(* IEC 61131-3 sources: Fosela-House-/control/lib, 8 files *)

(* ---- Types_Common.st ---- *)
(* ============================================================
   Types_Common.st
   Tipos, enumeraciones y constantes compartidos entre
   FREE Smart (solar) y FREE Evolution (sistema principal).
   Proyecto: Fusela House — Jerez de la Frontera
   ============================================================ *)

(* ------------------------------------------------------------
   ENUMERACIONES
   ------------------------------------------------------------ *)

(* Modos del subsistema solar *)
TYPE E_Solar_Mode :
(
    SOLAR_AUTO      := 0,   (* Lógica automática según temperaturas *)
    SOLAR_FORCE_ACS := 1,   (* Forzar desvío a ACS *)
    SOLAR_FORCE_POOL:= 2,   (* Forzar desvío a piscina *)
    SOLAR_OFF       := 3    (* Solar desactivado *)
);
END_TYPE

(* Destino del primario de la BDC *)
TYPE E_BDC_Mode :
(
    BDC_OFF         := 0,
    BDC_ACS         := 1,   (* V3V1→D2 *)
    BDC_CLIMATE     := 2,   (* V3V1→V3V2→D3 *)
    BDC_POOL        := 3    (* V3V1→V3V2→HX_BDC *)
);
END_TYPE

(* Destino del HTR *)
TYPE E_HTR_Mode :
(
    HTR_ACS         := 0,   (* V3V3→serp.sup D2 (por defecto) *)
    HTR_POOL        := 1    (* V3V3→HX_HTR *)
);
END_TYPE

(* Estado de válvula de 3 vías *)
TYPE E_Valve3Way_Pos :
(
    V3W_POS_A       := 0,   (* Posición A (desenergizada / muelle) *)
    V3W_POS_B       := 1    (* Posición B (energizada) *)
);
END_TYPE

(* Modo de apartamento *)
TYPE E_Apartment_Mode :
(
    APT_PRECALENTADA := 0,  (* Alimenta CE desde agua precalentada (por defecto) *)
    APT_AFS          := 1   (* Alimenta CE desde AFS directa *)
);
END_TYPE

(* Fases del ciclo de pasteurización *)
TYPE E_Pasteurization_Phase :
(
    PAST_IDLE        := 0,  (* Sin ciclo activo *)
    PAST_HEAT_D2     := 1,  (* Calentando D2 a 70 °C *)
    PAST_HOLD_D2     := 2,  (* Manteniendo D2 ≥ 70 °C durante t_hold *)
    PAST_FLUSH_APT   := 3,  (* Purgado secuencial de apartamentos *)
    PAST_DONE        := 4   (* Ciclo completado *)
);
END_TYPE

(* Prioridad de la BDC *)
TYPE E_BDC_Priority :
(
    PRIO_ACS_CLIMATE_POOL := 0,  (* ACS > Climatización > Piscina *)
    PRIO_ACS_POOL_CLIMATE := 1   (* ACS > Piscina > Climatización *)
);
END_TYPE

(* ------------------------------------------------------------
   ESTRUCTURAS
   ------------------------------------------------------------ *)

(* Datos del subsistema solar publicados por FREE Smart *)
TYPE ST_SolarData :
STRUCT
    TT1             : REAL;     (* Temperatura colector [°C] *)
    TT2             : REAL;     (* D1 fondo [°C] *)
    TT3             : REAL;     (* D1 cabeza [°C] *)
    DT_solar        : REAL;     (* ΔT medido TT1-TT2 [K] *)
    vel_P1          : UINT;     (* Velocidad P1 [0-1000 ‰] *)
    pos_V3V_SOL     : BOOL;     (* FALSE=ACS, TRUE=piscina *)
    persianas_cerradas : BOOL;
    P2_activo       : BOOL;
    alarma_solar    : UINT;     (* 0=OK, ver códigos *)
    comm_ok         : BOOL;     (* Comunicación Modbus activa *)
END_STRUCT
END_TYPE

(* Alarmas del sistema *)
TYPE ST_SystemAlarms :
STRUCT
    (* Solar *)
    ALM_TT1_HIGH        : BOOL;  (* TT1 > ALM_TT1_MAX *)
    ALM_TT2_HIGH        : BOOL;  (* TT2 > ALM_TT2_MAX *)
    ALM_COMM_SMART      : BOOL;  (* Pérdida comunicación FREE Smart *)
    (* ACS *)
    ALM_TT5_LOW         : BOOL;  (* D2 cabeza por debajo de mínimo *)
    ALM_TT5_HIGH        : BOOL;  (* D2 sobretemperatura *)
    (* Piscina *)
    ALM_PISC_FLUJO      : BOOL;  (* IF_PISC sin flujo durante calentamiento *)
    ALM_PISC_T_HIGH     : BOOL;  (* TT11 > máximo piscina *)
    (* Climatización *)
    ALM_INUNDACION      : BOOL;  (* Sensor inundación bandeja fancoil *)
    ALM_D3_HIGH         : BOOL;  (* D3 sobretemperatura *)
    (* General *)
    ALM_BDC_FAULT       : BOOL;  (* Fallo BDC (entrada digital) *)
    CUALQUIER_ALARMA    : BOOL;  (* OR de todas *)
END_STRUCT
END_TYPE

(* ------------------------------------------------------------
   CONSTANTES — TEMPERATURAS (°C)
   ------------------------------------------------------------ *)
VAR_GLOBAL CONSTANT

    (* Solar *)
    C_SOLAR_DT_START    : REAL := 6.0;   (* ΔT arranque P1 *)
    C_SOLAR_DT_STOP     : REAL := 3.0;   (* ΔT parada P1 *)
    C_SOLAR_DT_TARGET   : REAL := 8.0;   (* ΔT objetivo lazo PI *)
    C_SOLAR_TT3_POOL    : REAL := 75.0;  (* TT3 mínimo para desvío a piscina *)
    C_SOLAR_TT1_MAX     : REAL := 95.0;  (* Alarma sobretemperatura colector *)
    C_SOLAR_TT2_DISS    : REAL := 85.0;  (* TT2 máximo antes de disipación *)
    C_SOLAR_TT2_LEGIONELLA : REAL := 45.0; (* Si TT2 lleva días por debajo → arranque forzado *)

    (* ACS *)
    C_ACS_TT4_START     : REAL := 50.0;  (* TT4 D2 fondo — arranque carga BDC *)
    C_ACS_TT4_STOP      : REAL := 55.0;  (* TT4 D2 fondo — parada carga BDC *)
    C_ACS_TT5_TARGET    : REAL := 65.0;  (* TT5 D2 cabeza — setpoint ACS *)
    C_ACS_TT5_HYST      : REAL := 3.0;   (* Histéresis TT5 *)
    C_ACS_VMT1          : REAL := 55.0;  (* Temperatura VMT1 [°C] — ajuste físico *)
    C_ACS_PAST_TARGET   : REAL := 70.0;  (* Temperatura pasteurización D2 *)
    C_ACS_PAST_HYST     : REAL := 2.0;   (* Histéresis pasteurización *)
    C_ACS_HTR_TT5_STOP  : REAL := 68.0;  (* TT5 que inhibe HTR hacia D2 *)

    (* Climatización *)
    C_CLIM_HEAT_START   : REAL := 45.0;  (* TT6 D3 arranque calefacción BDC *)
    C_CLIM_HEAT_STOP    : REAL := 50.0;  (* TT6 D3 parada calefacción *)
    C_CLIM_COOL_START   : REAL := 9.0;   (* TT7 D3 arranque refrigeración *)
    C_CLIM_COOL_STOP    : REAL := 7.0;   (* TT7 D3 parada refrigeración *)

    (* Piscina *)
    C_POOL_TARGET       : REAL := 27.0;  (* TT11 setpoint temperatura piscina *)
    C_POOL_HYST         : REAL := 1.0;   (* Histéresis piscina *)
    C_POOL_MAX          : REAL := 32.0;  (* TT11 máximo — alarma *)

    (* Alarmas hardware *)
    C_ALM_TT1_MAX       : REAL := 95.0;
    C_ALM_TT2_MAX       : REAL := 88.0;  (* TK1 termostato hardware ≈ 88°C *)
    C_ALM_TT5_MAX       : REAL := 92.0;  (* Z2 hardware ≈ 95°C *)

END_VAR

(* ------------------------------------------------------------
   CONSTANTES — TIEMPOS
   ------------------------------------------------------------ *)
VAR_GLOBAL CONSTANT

    C_SOLAR_MIN_ON_TIME     : TIME := T#30S;   (* Tiempo mínimo P1 encendida *)
    C_SOLAR_MIN_OFF_TIME    : TIME := T#20S;   (* Tiempo mínimo P1 apagada *)
    C_VALVE_TRAVEL_TIME     : TIME := T#30S;   (* Tiempo de maniobra V3V *)
    C_MODBUS_POLL_PERIOD    : TIME := T#5S;    (* Periodo polling Modbus maestro *)
    C_MODBUS_TIMEOUT        : TIME := T#15S;   (* Timeout comunicación *)
    C_PAST_HOLD_TIME        : TIME := T#60M;   (* Tiempo mantenimiento pasteurización *)
    C_PAST_FLUSH_TIME       : TIME := T#30M;   (* Tiempo purgado por apartamento *)
    C_ALM_FILTER_TIME       : TIME := T#10S;   (* Filtro antirrebote alarmas *)
    C_LEGIONELLA_MAX_DAYS   : TIME := T#168H;  (* 7 días sin llegar a 60°C en TT2 *)
    C_VACANCIA_THRESHOLD    : TIME := T#336H;  (* 14 días → cambiar APT a AFS *)

END_VAR

(* ------------------------------------------------------------
   CONSTANTES — MODBUS REGISTROS
   (FREE Smart esclavo dirección 1)
   ------------------------------------------------------------ *)
VAR_GLOBAL CONSTANT

    (* Registros de lectura (FREE Smart → FREE Evolution) *)
    MB_REG_TT1          : UINT := 100;
    MB_REG_TT2          : UINT := 101;
    MB_REG_TT3          : UINT := 102;
    MB_REG_VEL_P1       : UINT := 103;
    MB_REG_EST_V3VSOL   : UINT := 104;
    MB_REG_EST_PERS     : UINT := 105;
    MB_REG_EST_P2       : UINT := 106;
    MB_REG_ALM_SOLAR    : UINT := 107;
    MB_REG_DT_SOLAR     : UINT := 108;

    (* Registros de escritura (FREE Evolution → FREE Smart) *)
    MB_REG_SP_DT        : UINT := 200;
    MB_REG_MODO_SOLAR   : UINT := 201;
    MB_REG_ORD_PERS     : UINT := 202;
    MB_REG_SP_TT3_POOL  : UINT := 203;

    (* Escala para valores de temperatura en Modbus (×10) *)
    MB_TEMP_SCALE       : REAL := 10.0;

    (* Dirección esclavo FREE Smart *)
    MB_SMART_SLAVE_ADDR : UINT := 1;

END_VAR

(* ---- GVL_Params.st ---- *)
(* ============================================================
   GVL_Params.st  –  Todos los parámetros Pnn del sistema
   RETAIN: sobreviven a corte de alimentación.
   Editables desde HMI según nivel de acceso (CFG / L1).
   Los rangos [Mín–Máx] se validan en runtime respecto a P00-P06.
   ============================================================ *)

VAR_GLOBAL RETAIN

    (* ── P00-P06  Límites de equipo (CFG) ───────────────────
       Introducir en puesta en marcha con datos de placa.
       No tienen defecto numérico: el instalador los introduce. *)
    P00_AccumulatorMaxTemp    : REAL := 0.0;  (* P00 *)
    P01_BDCMaxFlowTemp        : REAL := 0.0;  (* P01 *)
    P02_HTRMaxTemp            : REAL := 0.0;  (* P02 *)
    P03_BDCMinCoolTemp        : REAL := 0.0;  (* P03 *)
    P04_CollectorMaxOperTemp  : REAL := 0.0;  (* P04 *)
    P05_HXMaxTemp             : REAL := 0.0;  (* P05 *)
    P06_PumpMaxFluidTemp      : REAL := 0.0;  (* P06 *)

    (* ── P10-P19  Solar (L1) ─────────────────────────────── *)
    P10_SolarDeltaTTarget          : REAL := 8.0;   (* P10  K *)
    P11_SolarDeltaTStart           : REAL := 6.0;   (* P11  K *)
    P12_SolarDeltaTStop            : REAL := 3.0;   (* P12  K *)
    P13_SolarPumpMinSpeed          : REAL := 10.0;  (* P13  % *)
    P14_SolarPumpMinOnTime         : TIME := T#30S; (* P14 *)
    P15_SolarPumpMinOffTime        : TIME := T#20S; (* P15 *)
    P16_MinTempForPoolSolarHeating : REAL := 75.0;  (* P16  °C *)
    P17_SolarOverheatShutterClose  : REAL := 85.0;  (* P17  °C *)
    P18_SolarOverheatShutterHyst   : REAL := 4.0;   (* P18  K *)
    P19_SolarMode                  : UINT := 0;     (* P19  0=AUTO *)

    (* ── P20-P23  Reguladores PI — solar y ACS (CFG) ───────
       Kp/Ki a ajustar en puesta en marcha tras análisis de respuesta.
       Valores iniciales conservadores. *)
    P20_SolarPI_Kp  : REAL := 0.50;  (* P20  adimensional CFG *)
    P21_SolarPI_Ki  : REAL := 0.08;  (* P21  1/s             CFG *)
    P22_DHWPI_Kp    : REAL := 0.40;  (* P22  adimensional CFG *)
    P23_DHWPI_Ki    : REAL := 0.05;  (* P23  1/s             CFG *)

    (* ── P30-P39  Estación producción ACS al paso (L1/CFG) ─
       P30-P31: reservorio (fuente de energía primaria)
       P32-P35: intercambiador de placas y control
       P36-P39: instrumentación y bomba PWM1 *)
    P30_DHWReservoirSetPoint      : REAL := 70.0;   (* P30  °C  setpoint carga reservorio   L1  *)
    P31_DHWReservoirHysteresis    : REAL := 4.0;    (* P31  K   histéresis carga            L1  *)
    P32_DHWReservoirMinForACS     : REAL := 65.0;   (* P32  °C  mín. reservorio para prod.  CFG *)
    P33_DHWReservoirAlarmLow      : REAL := 60.0;   (* P33  °C  alarma reservorio frío      CFG *)
    P34_DHWPlateOutputSetpoint    : REAL := 60.0;   (* P34  °C  consigna salida placa       L1  *)
    P35_DHWPlateOutputHysteresis  : REAL := 2.0;    (* P35  K   histéresis control PI       CFG *)
    P36_DHWFlowMeterK             : REAL := 6.6;    (* P36  pulsos/L·min  K caudalímetro    CFG — confirmar ficha YF-B6 *)
    P37_DHWFlowDetectMin          : REAL := 0.5;    (* P37  L/min  umbral detección grifo   CFG *)
    P38_DHWPumpCooldown           : TIME  := T#15S; (* P38  s     tiempo post-cierre grifo  CFG *)
    P39_DHWMaxOutputAlarm         : REAL := 68.0;   (* P39  °C  alarma sobretemperatura ACS CFG *)

    (* ── P40-P46  ACS apartamentos (L1) ─────────────────── *)
    P40_AptMode_01       : UINT := 0;     (* P40  0=PREC 1=AFS *)
    P41_AptMode_02       : UINT := 0;     (* P41 *)
    P42_AptMode_03       : UINT := 0;     (* P42 *)
    P43_AptMode_04       : UINT := 0;     (* P43 *)
    P44_AptMode_05       : UINT := 0;     (* P44 *)

    (* ── P50-P53  Climatización (L1) ────────────────────── *)
    P50_HeatingSetPoint  : REAL := 45.0;  (* P50  °C *)
    P51_HeatingHysteresis: REAL := 4.0;   (* P51  K *)
    P52_CoolingSetPoint  : REAL := 9.0;   (* P52  °C *)
    P53_CoolingHysteresis: REAL := 2.0;   (* P53  K *)

    (* ── P54-P57  Clima reversible y muestreo solar (CFG) ──
       NADA HARDCODED: enclavamiento estacional y muestreo a bajo caudal *)
    P54_SeasonChangeMinHold : TIME := T#10M;  (* P54  histéresis temporal de cambio de estación *)
    P55_SeasonInterlockDelay: TIME := T#20S;  (* P55  retardo válvulas-en-posición antes de bombas *)
    P56_SolarSampleInterval : TIME := T#15M;  (* P56  cada cuánto se muestrea el campo solar *)
    P57_SolarSampleDuration : TIME := T#90S;  (* P57  duración ventana de muestreo a bajo caudal *)

    (* ── P60-P64  Piscina (L1) ──────────────────────────── *)
    P60_PoolSetPoint         : REAL := 27.0;   (* P60  °C *)
    P61_PoolHysteresis       : REAL := 1.0;    (* P61  K *)
    P62_PoolMaxTemp          : REAL := 32.0;   (* P62  °C *)
    P63_PoolDelay            : TIME := T#30S;  (* P63 *)
    P64_PoolValveTravelTime  : TIME := T#15S;  (* P64 *)

    (* ── P70-P77  Higienización (L1/CFG) ────────────────── *)
    P70_PreheatingTarget      : REAL := 70.0;    (* P70  °C  L1 *)
    P71_PreheatingHysteresis  : REAL := 2.0;     (* P71  K   L1 *)
    P72_PreheatingHoldTime    : TIME := T#60M;   (* P72       L1 *)
    P73_PreheatingFlushTime   : TIME := T#30M;   (* P73       L1 *)
    P74_PreheatingDayOfWeek   : UINT := 1;       (* P74  1=Lun L1 *)
    P75_PreheatingHour        : UINT := 3;       (* P75  hora L1 *)
    P76_D1PreheatingMaxDays   : UINT := 7;       (* P76  días CFG *)
    P77_D1PreheatingMinTemp   : REAL := 60.0;    (* P77  °C  CFG *)

    (* ── P80  Prioridades (CFG) ──────────────────────────── *)
    P80_BDCPriority : UINT := 0;  (* P80  0=ACS>CLIM>PISC *)

    (* ── P90-P97  Sistema / Modbus / HMI (CFG) ──────────── *)
    P90_ModbusSlaveAddr  : UINT := 1;     (* P90 *)
    P91_ModbusBaudrate   : UINT := 1;     (* P91  1=19200 *)
    P92_ModbusPollPeriod : TIME := T#5S;  (* P92 *)
    P93_ModbusTimeout    : TIME := T#15S; (* P93 *)
    P94_PIN_L1           : UINT := 1234;  (* P94 *)
    P95_PIN_CFG          : UINT := 9999;  (* P95 *)
    P96_PIN_MaxAttempts  : UINT := 3;     (* P96 *)
    P97_SessionTimeout   : TIME := T#10M; (* P97 *)

    (* ── OS00-OS13  Offsets de sondas (CFG) ─────────────── *)
    OS00_TT1  : REAL := 0.0;  (* OS00  K *)
    OS01_TT2  : REAL := 0.0;  (* OS01 *)
    OS02_TT3  : REAL := 0.0;  (* OS02 *)
    OS03_TT4  : REAL := 0.0;  (* OS03 *)
    OS04_TT5  : REAL := 0.0;  (* OS04 *)
    OS05_TT6  : REAL := 0.0;  (* OS05 *)
    OS06_TT7  : REAL := 0.0;  (* OS06 *)
    OS07_TT8  : REAL := 0.0;  (* OS07 *)
    OS08_TT9  : REAL := 0.0;  (* OS08 *)
    OS00_TT10 : REAL := 0.0;  (* OS09 *)
    OS00_TT11 : REAL := 0.0;  (* OS10 *)
    OS00_TT12 : REAL := 0.0;  (* OS11 *)
    OS00_TT13 : REAL := 0.0;  (* OS12 *)
    OS00_TT14 : REAL := 0.0;  (* OS13 *)

END_VAR

(* ---- FB_Alarm.st ---- *)
(* ============================================================
   FB_Alarm.st
   Alarma con filtro antirrebote, enclavamiento (latch) y reset.
   - filter_time: la condición debe persistir antes de activar alarma.
   - Latch: una vez activa, se mantiene hasta reset explícito.
   ============================================================ *)

FUNCTION_BLOCK FB_Alarm

VAR_INPUT
    condition       : BOOL;             (* TRUE = condición de alarma *)
    reset_cmd       : BOOL;             (* Pulso → desenclavamiento *)
    filter_time     : TIME := T#10S;    (* Tiempo de filtrado *)
    latch           : BOOL := TRUE;     (* TRUE = enclavamiento activo *)
    enabled         : BOOL := TRUE;
END_VAR

VAR_OUTPUT
    active          : BOOL;             (* Alarma activa (enclavada si latch) *)
    pending         : BOOL;             (* Condición presente pero no enclavada aún *)
END_VAR

VAR
    timer_filter    : TON;
    latched         : BOOL := FALSE;
END_VAR

(* --- Implementación --- *)

IF NOT enabled THEN
    active  := FALSE;
    pending := FALSE;
    latched := FALSE;
    timer_filter(IN := FALSE, PT := filter_time);
    RETURN;
END_IF

(* Filtro antirrebote *)
timer_filter(IN := condition, PT := filter_time);
pending := condition AND NOT timer_filter.Q;

(* Enclavamiento *)
IF timer_filter.Q THEN
    latched := TRUE;
END_IF

IF reset_cmd AND NOT condition THEN
    latched := FALSE;
END_IF

IF latch THEN
    active := latched;
ELSE
    active := timer_filter.Q;
END_IF

END_FUNCTION_BLOCK

(* ---- FB_Hysteresis.st ---- *)
(* ============================================================
   FB_Hysteresis.st
   Control todo-nada con histéresis configurable.
   Reutilizado en: ACS, climatización, piscina, persianas.

   Ejemplo de uso:
     ctrl_TT5(
       measured    := TT5,
       setpoint    := C_ACS_TT5_TARGET,
       hysteresis  := C_ACS_TT5_HYST,
       mode_heat   := TRUE   (* TRUE=calor: ON si T<SP; FALSE=frío: ON si T>SP *)
     );
     output_device := ctrl_TT5.output;
   ============================================================ *)

FUNCTION_BLOCK FB_Hysteresis

VAR_INPUT
    measured    : REAL;         (* Valor medido *)
    setpoint    : REAL;         (* Consigna *)
    hysteresis  : REAL;         (* Banda muerta total [mismas unidades que measured] *)
    mode_heat   : BOOL := TRUE; (* TRUE=modo calor (ON si T<SP); FALSE=modo frío (ON si T>SP) *)
    enabled     : BOOL := TRUE; (* FALSE inhibe la salida (→ FALSE) *)
END_VAR

VAR_OUTPUT
    output      : BOOL;         (* Salida de control *)
    error       : REAL;         (* SP - measured *)
END_VAR

VAR
    half_hyst   : REAL;
END_VAR

(* --- Implementación --- *)

error    := setpoint - measured;
half_hyst := hysteresis / 2.0;

IF NOT enabled THEN
    output := FALSE;

ELSIF mode_heat THEN
    (* Modo calor: activa cuando T cae por debajo de (SP - H/2) *)
    IF measured <= (setpoint - half_hyst) THEN
        output := TRUE;
    ELSIF measured >= (setpoint + half_hyst) THEN
        output := FALSE;
    END_IF
    (* Entre las dos bandas: mantiene estado anterior *)

ELSE
    (* Modo frío: activa cuando T sube por encima de (SP + H/2) *)
    IF measured >= (setpoint + half_hyst) THEN
        output := TRUE;
    ELSIF measured <= (setpoint - half_hyst) THEN
        output := FALSE;
    END_IF

END_IF

END_FUNCTION_BLOCK

(* ---- FB_PI_Controller.st ---- *)
(* ============================================================
   FB_PI_Controller.st
   Controlador PI discreto con anti-windup y saturación.
   Usado para: bomba solar P1 (lazo ΔT constante).

   Salida: 0.0 – 100.0 (%) que el caller mapea a 0-10V / 0-1000‰
   ============================================================ *)

FUNCTION_BLOCK FB_PI_Controller

VAR_INPUT
    measured        : REAL;         (* Valor medido (ej: ΔT actual) *)
    setpoint        : REAL;         (* Consigna (ej: ΔT objetivo 8 K) *)
    Kp              : REAL := 0.5;  (* Ganancia proporcional *)
    Ki              : REAL := 0.08; (* Ganancia integral [1/s] *)
    out_min         : REAL := 0.0;  (* Límite inferior salida [%] *)
    out_max         : REAL := 100.0;(* Límite superior salida [%] *)
    dt_seconds      : REAL := 1.0;  (* Periodo de muestreo [s] — igualar al task cycle *)
    enabled         : BOOL := TRUE; (* FALSE → salida a out_min, integral a 0 *)
    reset           : BOOL := FALSE;(* Pulso → resetea integral *)
END_VAR

VAR_OUTPUT
    output          : REAL;         (* Salida [out_min..out_max] *)
    error           : REAL;         (* Setpoint - measured *)
    saturated       : BOOL;         (* TRUE si la salida está saturada *)
END_VAR

VAR
    integral        : REAL := 0.0;
    p_term          : REAL;
    i_term          : REAL;
    raw_output      : REAL;
END_VAR

(* --- Implementación --- *)

IF reset THEN
    integral := 0.0;
END_IF

IF NOT enabled THEN
    output   := out_min;
    integral := 0.0;
    saturated := FALSE;
    error    := 0.0;
    RETURN;
END_IF

error  := setpoint - measured;
p_term := Kp * error;

(* Anti-windup: solo integra si la salida no está saturada
   (o si el error va en dirección opuesta a la saturación) *)
IF NOT saturated OR
   (saturated AND ((output >= out_max AND error < 0.0) OR
                   (output <= out_min AND error > 0.0))) THEN
    integral := integral + Ki * error * dt_seconds;
END_IF

raw_output := p_term + integral;

(* Saturación de salida *)
IF raw_output > out_max THEN
    output    := out_max;
    saturated := TRUE;
ELSIF raw_output < out_min THEN
    output    := out_min;
    saturated := TRUE;
ELSE
    output    := raw_output;
    saturated := FALSE;
END_IF

END_FUNCTION_BLOCK

(* ---- FB_Pump.st ---- *)
(* ============================================================
   FB_Pump.st
   Gestión de bomba/circuladora con:
   - Tiempo mínimo encendida (anti-ciclado)
   - Tiempo mínimo apagada (anti-ciclado)
   - Inhibición por alarma
   Reutilizado en: P1, P2, P3, P4
   ============================================================ *)

FUNCTION_BLOCK FB_Pump

VAR_INPUT
    cmd_run         : BOOL;             (* TRUE = orden de marcha *)
    fault           : BOOL := FALSE;    (* TRUE = fallo externo → parada forzada *)
    min_on_time     : TIME := T#30S;    (* Tiempo mínimo encendida *)
    min_off_time    : TIME := T#20S;    (* Tiempo mínimo apagada *)
    enabled         : BOOL := TRUE;
END_VAR

VAR_OUTPUT
    DO_pump         : BOOL;             (* Señal física *)
    running         : BOOL;             (* Confirmación de marcha *)
    inhibited       : BOOL;             (* TRUE si en periodo de inhibición *)
END_VAR

VAR
    timer_min_on    : TON;
    timer_min_off   : TON;
    internal_run    : BOOL := FALSE;
END_VAR

(* --- Implementación --- *)

IF NOT enabled OR fault THEN
    internal_run := FALSE;
    DO_pump      := FALSE;
    running      := FALSE;
    inhibited    := FALSE;
    timer_min_on(IN := FALSE, PT := min_on_time);
    timer_min_off(IN := FALSE, PT := min_off_time);
    RETURN;
END_IF

(* Timer anti-ciclado apagado: una vez parada no vuelve a arrancar hasta cumplir min_off *)
timer_min_off(IN := NOT internal_run, PT := min_off_time);

(* Arranque: cmd_run activo Y periodo mínimo de parada cumplido *)
IF cmd_run AND (timer_min_off.Q OR internal_run) THEN
    internal_run := TRUE;
END_IF

(* Timer anti-ciclado encendido: una vez arrancada no para hasta cumplir min_on *)
timer_min_on(IN := internal_run, PT := min_on_time);

(* Parada: cmd_run inactivo Y periodo mínimo de marcha cumplido *)
IF NOT cmd_run AND timer_min_on.Q THEN
    internal_run := FALSE;
END_IF

DO_pump  := internal_run;
running  := internal_run;
inhibited := (cmd_run AND NOT timer_min_off.Q AND NOT internal_run) OR
             (NOT cmd_run AND NOT timer_min_on.Q AND internal_run);

END_FUNCTION_BLOCK

(* ---- FB_Valve2Way.st ---- *)
(* ============================================================
   FB_Valve2Way.st
   Gestión de válvula motorizada 2 vías todo-nada.
   - Tiempo mínimo de apertura para proteger el actuador.
   - Reutilizado en: VP_HX1, VP_HX_BDC, VP_HX_HTR
   ============================================================ *)

FUNCTION_BLOCK FB_Valve2Way

VAR_INPUT
    cmd_open        : BOOL;             (* TRUE = abrir *)
    enabled         : BOOL := TRUE;     (* FALSE fuerza cierre *)
    min_open_time   : TIME := T#10S;    (* Tiempo mínimo apertura *)
    travel_time     : TIME := T#15S;    (* Tiempo de maniobra *)
END_VAR

VAR_OUTPUT
    DO_valve        : BOOL;             (* Señal física al actuador *)
    is_open         : BOOL;             (* Confirmación apertura *)
    in_transit      : BOOL;
END_VAR

VAR
    timer_min       : TON;
    timer_travel    : TON;
    last_cmd        : BOOL := FALSE;
END_VAR

(* --- Implementación --- *)

IF NOT enabled THEN
    DO_valve   := FALSE;
    is_open    := FALSE;
    in_transit := FALSE;
    timer_min(IN := FALSE, PT := min_open_time);
    timer_travel(IN := FALSE, PT := travel_time);
    last_cmd := FALSE;
    RETURN;
END_IF

(* Tiempo mínimo de apertura: una vez abierta no cierra hasta cumplir min_open_time *)
IF cmd_open AND NOT last_cmd THEN
    timer_min(IN := FALSE, PT := min_open_time);
END_IF
timer_min(IN := DO_valve, PT := min_open_time);

(* Comando efectivo: abre si cmd_open, o mantiene abierto durante min_open_time *)
DO_valve := (cmd_open AND enabled) OR (timer_min.Q = FALSE AND DO_valve AND enabled);

(* Confirmar cambio de estado → in_transit *)
IF DO_valve <> last_cmd THEN
    in_transit := TRUE;
    timer_travel(IN := FALSE, PT := travel_time);
END_IF
last_cmd := DO_valve;

timer_travel(IN := in_transit, PT := travel_time);
IF timer_travel.Q THEN
    in_transit := FALSE;
    timer_travel(IN := FALSE, PT := travel_time);
END_IF

is_open := DO_valve AND NOT in_transit;

END_FUNCTION_BLOCK

(* ---- FB_Valve3Way.st ---- *)
(* ============================================================
   FB_Valve3Way.st
   Gestión de válvula motorizada 3 vías todo-nada.
   - Protege contra cambios de posición durante la maniobra.
   - Salida: DO_valve = FALSE → posición A (muelle/reposo)
             DO_valve = TRUE  → posición B (energizada)
   - Reutilizado en: V3V1, V3V2, V3V3, V3V_SOL
   ============================================================ *)

FUNCTION_BLOCK FB_Valve3Way

VAR_INPUT
    cmd_pos_B       : BOOL;             (* TRUE = ir a posición B *)
    enabled         : BOOL := TRUE;     (* FALSE fuerza posición A *)
    travel_time     : TIME := T#30S;    (* Tiempo de maniobra *)
END_VAR

VAR_OUTPUT
    DO_valve        : BOOL;             (* Señal física al actuador *)
    position        : E_Valve3Way_Pos;  (* Posición confirmada *)
    in_transit      : BOOL;             (* TRUE durante maniobra *)
END_VAR

VAR
    timer_travel    : TON;
    last_cmd        : BOOL := FALSE;
    target          : BOOL := FALSE;
END_VAR

(* --- Implementación --- *)

IF NOT enabled THEN
    DO_valve    := FALSE;
    position    := V3W_POS_A;
    in_transit  := FALSE;
    last_cmd    := FALSE;
    timer_travel(IN := FALSE, PT := travel_time);
    RETURN;
END_IF

target := cmd_pos_B;

(* Detecta cambio de comando *)
IF target <> last_cmd THEN
    timer_travel(IN := FALSE, PT := travel_time); (* Reinicia timer *)
    in_transit := TRUE;
    last_cmd   := target;
END_IF

(* Temporizador de maniobra *)
timer_travel(IN := in_transit, PT := travel_time);

IF timer_travel.Q THEN
    in_transit := FALSE;
    timer_travel(IN := FALSE, PT := travel_time);
END_IF

(* Salida física *)
DO_valve := target;

(* Posición confirmada solo cuando no está en maniobra *)
IF NOT in_transit THEN
    IF DO_valve THEN
        position := V3W_POS_B;
    ELSE
        position := V3W_POS_A;
    END_IF
END_IF

END_FUNCTION_BLOCK
